FUNCTION_BLOCK TE_AxisBasic_V2
VAR_INPUT
END_VAR

VAR_OUTPUT
END_VAR

VAR
    PowerControl :MC_Power;
    bAxisEnable  :BOOL;
	{attribute 'no_copy'}
    AdminCtrl      :REFERENCE TO ST_AXIS_ADMINISTRATION;
	{attribute 'no_copy'}
    PosModeCtrl    :REFERENCE TO ST_AXIS_POSITION;
	{attribute 'no_copy'}
    VelModeCtrl    :REFERENCE TO ST_AXIS_VELOCITY;
	{attribute 'no_copy'}
    SyncModeCtrl   :REFERENCE TO ST_AXIS_SYNCHRONISATION;
	{attribute 'no_copy'}
    TorqueModeCtrl :REFERENCE TO ST_AXIS_TORQUE;
	{attribute 'no_copy'}
    SetupModeCtrl  :REFERENCE TO ST_AXIS_SETUP_MODE;
	{attribute 'no_copy'}
	AdminStatus : REFERENCE TO ST_AXIS_ADMIN_STATUS;
	{attribute 'no_copy'}
	DiagStatus : REFERENCE TO ST_AXIS_DIAGNOSIS;
	{attribute 'no_copy'}
	PosModeStatus : REFERENCE TO ST_AXIS_POS_STATUS;
	{attribute 'no_copy'}
	VelModeStatus : REFERENCE TO ST_AXIS_VEL_STATUS;
	{attribute 'no_copy'}
	SyncModeStatus: REFERENCE TO ST_AXIS_SYNC_STATUS;
	{attribute 'no_copy'}
	SetupModeStatus: REFERENCE TO ST_AXIS_SETUP_MODE_STATUS;
	ClearError: MC_Reset;
	bAxisStop: BOOL;
END_VAR


//=========================================//
// Cyclic update						   //
//=========================================//
A90_Cyclic();

ACTION A00_ModeAb:
// Check Reference available
IF NOT __ISVALIDREF(AdminCtrl) THEN
	RETURN;
END_IF

// Check Operation mode is ModeAb
IF AdminCtrl._OpMode.en <> ModeAb THEN
	RETURN;
END_IF

// Check Axis Servo OFF
IF NOT  AdminCtrl.Axis.Status.Disabled THEN
	AdminStatus.ModeAb := TRUE;
	AdminStatus._OpModeAck := ModeAb;
	AdminStatus.CmdDone := TRUE;
END_IF
END_ACTION

ACTION A01_ModeAH:
IF AdminCtrl._OpMode.en <> ModeAH THEN
	RETURN;
END_IF

IF AdminCtrl.Axis.Status.StandStill THEN
	AdminCtrl.Axis.Status.
END_IF
END_ACTION

ACTION A90_Cyclic:
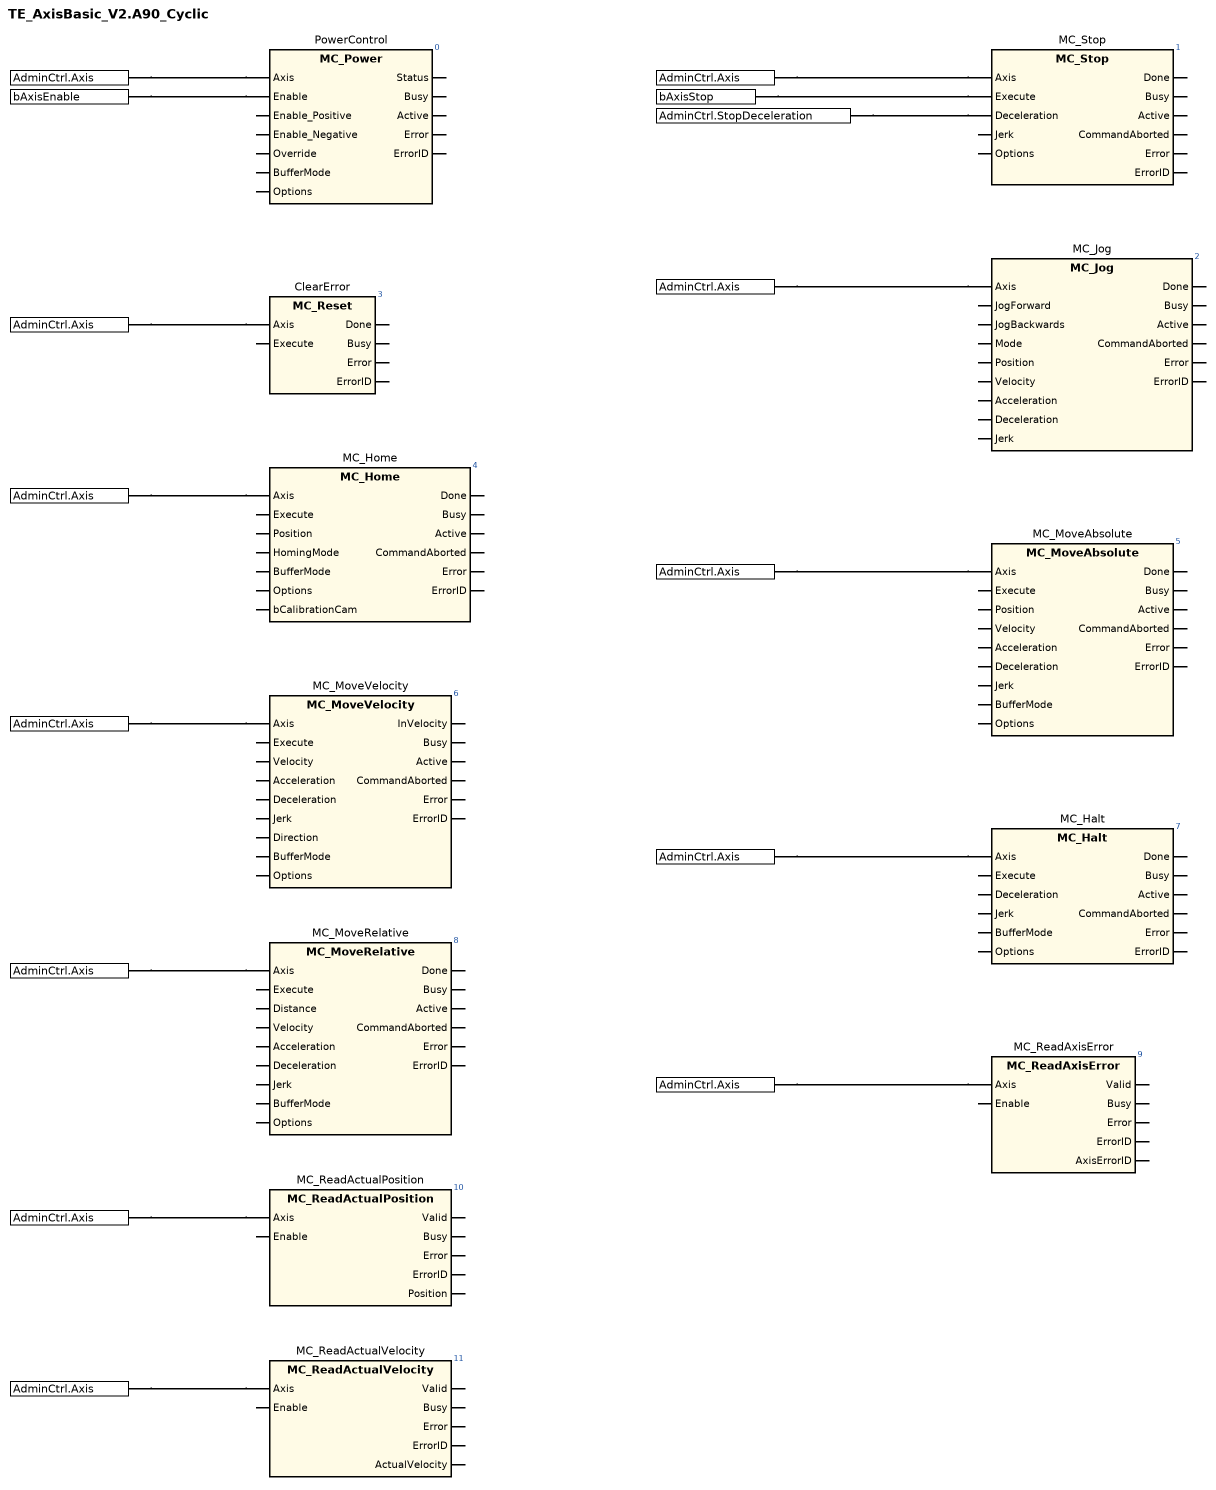
PowerControl(Axis := AdminCtrl.Axis, Enable := bAxisEnable); // MC_Power
MC_Stop(Axis := AdminCtrl.Axis, Execute := bAxisStop, Deceleration := AdminCtrl.StopDeceleration);
MC_Jog(Axis := AdminCtrl.Axis);
ClearError(Axis := AdminCtrl.Axis); // MC_Reset
MC_Home(Axis := AdminCtrl.Axis);
MC_MoveAbsolute(Axis := AdminCtrl.Axis);
MC_MoveVelocity(Axis := AdminCtrl.Axis);
MC_Halt(Axis := AdminCtrl.Axis);
MC_MoveRelative(Axis := AdminCtrl.Axis);
MC_ReadAxisError(Axis := AdminCtrl.Axis);
MC_ReadActualPosition(Axis := AdminCtrl.Axis);
MC_ReadActualVelocity(Axis := AdminCtrl.Axis);
END_ACTION

METHOD M_GetOpMode : E_AXIS_MODE
VAR_INPUT
END_VAR
IF __ISVALIDREF(AdminStatus) THEN
	M_GetOpMode := AdminStatus._OpModeAck;
END_IF
END_METHOD

METHOD M_InitExtension
VAR_INPUT
	Index : UINT;
END_VAR
//=============================================================//
//Reference access											   //
//=============================================================//
AdminCtrl      REF= arAxisCtrl_gb[Index].Admin;
PosModeCtrl    REF= arAxisCtrl_gb[Index].PosMode;
VelModeCtrl    REF= arAxisCtrl_gb[Index].VelMode;
SyncModeCtrl   REF= arAxisCtrl_gb[Index].SyncMode;
TorqueModeCtrl REF= arAxisCtrl_gb[Index].TorqueMode;
SetupModeCtrl  REF= arAxisCtrl_gb[Index].SetupMode;

AdminStatus     REF= arAxisStutus_gb[Index].Admin;
DiagStatus      REF= arAxisStutus_gb[Index].Diag;
PosModeStatus   REF= arAxisStutus_gb[Index].PosMode;
VelModeStatus   REF= arAxisStutus_gb[Index].VelMode;
SyncModeStatus  REF= arAxisStutus_gb[Index].SyncMode;
SetupModeStatus REF= arAxisStutus_gb[Index].SetupMode;
END_METHOD

END_FUNCTION_BLOCK

(* stored: Version 1.1.0.1, ProductVersion 3.1.4024.11
   POU TE_AxisBasic_V2: Id {1d96a586-d41c-4a71-88d9-3cca03df4dc2}, SpecialFunc None
   Action A00_ModeAb: Id {24ea519f-f158-457d-8209-e4bc50b8f442}
   Action A01_ModeAH: Id {8cffe33c-0d2a-41cd-87c6-44acc73e7032}
   Action A90_Cyclic: Id {6de0965f-b939-4e05-a93a-927519bdfb7c}
   Method M_GetOpMode: Id {ddd5da4b-8e59-48bf-aa86-349d80498a92}
   Method M_InitExtension: Id {28bd45e1-2c02-4b36-ada7-a127ff0171be} *)
